  MoveL speed 30 mm/s, acceleration 50 mm/s^2 (useActiveTCP=true optimoveEnabled=false optiMoveSpeed=0.3 optiMoveAcceleration=0.09) feature=Base
    SuppressedNode
      Waypoint r1_ek_front: TCP in base x=439.065 y=405.452 z=65.996 mm, rx=2.3168 ry=2.0514 rz=0.0766 rad; joints [-187.962, -93.321, 143.386, -27.168, -1.131, -26.752] deg
    SuppressedNode
      Waypoint r1_ek_middle: TCP in base x=419.01 y=404.851 z=65.995 mm, rx=2.3096 ry=2.0447 rz=0.0891 rad; joints [-188.553, -97.485, 146.002, -33.769, -1.69, -19.324] deg
    SuppressedNode
      Waypoint r1_ek_middle2: TCP in base x=417.012 y=405.435 z=65.003 mm, rx=2.3169 ry=2.0513 rz=0.0766 rad; joints [-188.493, -97.025, 145.794, -33.21, -1.638, -19.415] deg
    SuppressedNode
      Waypoint r1_ek_bottom: TCP in base x=413.072 y=405.431 z=68 mm, rx=2.3168 ry=2.0513 rz=0.0767 rad; joints [-188.596, -97.887, 146.02, -33.517, -1.738, -18.475] deg
    SuppressedNode
      Waypoint r1_ek_end: TCP in base x=389.999 y=405.444 z=68.005 mm, rx=2.3169 ry=2.0514 rz=0.0766 rad; joints [-189.248, -101.07, 148.002, -36.337, -2.38, -14.447] deg
    Waypoint Variable (Variable): variable=ek_front
    Waypoint Variable (Variable): variable=ek_middle
    Waypoint Variable (Variable): variable=ek_middle2
    Waypoint Variable (Variable): variable=ek_bottom
    Waypoint Variable (Variable): variable=ek_end
  MoveJ speed 60 deg/s, acceleration 80 deg/s^2 (useActiveTCP=true optimoveEnabled=false optiMoveSpeed=0.3 optiMoveAcceleration=0.09) feature=Base
    SuppressedNode
      Waypoint r1_ek_oldhome: TCP in base x=397.38 y=356.254 z=319.821 mm, rx=2.3163 ry=2.0576 rz=0.0741 rad; joints [-198.126, -117.851, 133.303, -13.009, -11.422, -6.035] deg
    Waypoint Variable (Variable): variable=ek_oldhome
    'above waypoint is home'
  SuppressedNode
    SafeHome (positionOptionType=SPEED_AND_ACCELERATION speed=1.047198 acceleration=1.396263 nextMotionTime=2)
SubProgram Straight_Homing_Floor_2 (keepSynchronizedWithDisk=false) programFile=/programs/Straight Homing Floor 2.urp
  Set NoAction tcp=pretend_w_top
  'dummy move below for debug'
  SuppressedNode
    Folder dummy points
      MoveL speed 100 mm/s, acceleration 1200 mm/s^2 (useActiveTCP=true optimoveEnabled=false optiMoveSpeed=0.3 optiMoveAcceleration=0.09) feature=Base
        Waypoint tcp_l: TCP in base x=-1157.117 y=-14.284 z=-81.871 mm, rx=1.2641 ry=-1.1744 rz=-0.9868 rad; joints [-20.789, -44.61, 126.749, -78.291, 59.56, 3.601] deg; TCP offset x=0.14 y=-17.51 z=284 mm, rx=0 ry=0 rz=0 rad
        Waypoint tcp_r: TCP in base x=-1091.012 y=400.793 z=-81.871 mm, rx=1.2641 ry=-1.1744 rz=-0.9868 rad; joints [-50.03, -43.105, 118.828, -69.165, 30.433, -0.106] deg
      tcp_pose_left := tcp_l
      tcp_pose_right := tcp_r
  SuppressedNode
    SafeHome (positionOptionType=SPEED_AND_ACCELERATION speed=1.047198 acceleration=1.396263 nextMotionTime=2)
  SuppressedNode
    MoveJ speed 60 deg/s, acceleration 80 deg/s^2 (useActiveTCP=true optimoveEnabled=false optiMoveSpeed=0.3 optiMoveAcceleration=0.09) feature=Base
      Waypoint demo_point0: TCP in base x=-1268.829 y=243.799 z=397.866 mm, rx=1.3918 ry=-0.5735 rz=-1.0174 rad; joints [-39.169, -62.377, 106.188, -68.476, 20.677, 9.969] deg; TCP offset x=-1.032 y=-18.062 z=285.234 mm, rx=0 ry=0 rz=0 rad
  SuppressedNode
    MoveJ speed 60 deg/s, acceleration 80 deg/s^2 (useActiveTCP=true optimoveEnabled=false optiMoveSpeed=0.3 optiMoveAcceleration=0.09) feature=Base
      Waypoint Waypoint_1: TCP in base x=-589.354 y=-224.033 z=519.728 mm, rx=1.0077 ry=-1.3585 rz=-1.2216 rad; joints [24.032, -118.039, 143.045, -26.295, 122.645, 7.654] deg
      Waypoint Waypoint_2: TCP in base x=-1013.668 y=283.774 z=13.404 mm, rx=-0.1302 ry=-1.6605 rz=-0.1403 rad; joints [-36.803, -53.188, 133.142, -74.065, 63.057, 86.565] deg; TCP offset x=0 y=0 z=246 mm, rx=0 ry=0 rz=0 rad
  Wait Sleep waitTime=1
  SuppressedNode
    tp := get_actual_tcp_pose()
  Script file /programs/analyze_touchpoints.script
    | (same text as the earlier copy of this file)
  path_pre := get_straight_homing_pathpoints_floor(tcp_pose_left,tcp_pose_right)
  ph1 := path_pre[0]
  ph2 := path_pre[1]
  ph3 := path_pre[2]
  ph4 := path_pre[3]
  ph4a := p[ph4[0]+0.1,ph4[1],ph4[2],ph4[3],ph4[4],ph4[5]]
  MoveL speed 250 mm/s, acceleration 1200 mm/s^2 (useActiveTCP=true optimoveEnabled=false optiMoveSpeed=0.3 optiMoveAcceleration=0.09) feature=Base
    MoveDirectionNode (selectedDirection=XPlus)
      Until DISTANCE (allowActions=false deceleration=3 distanceNodeType=STOP) Distance=0.1; motionParameters(blendRadius=0)
  SuppressedNode
    MoveJ speed 60 deg/s, acceleration 80 deg/s^2 (useActiveTCP=true optimoveEnabled=false optiMoveSpeed=0.3 optiMoveAcceleration=0.09) feature=Base
      SuppressedNode
        Waypoint Waypoint_11: TCP in base x=-589.354 y=-454.462 z=658.693 mm, rx=1.8664 ry=-1.8664 rz=-0.5984 rad; joints [32.16, -93.601, 92.579, 59.83, 108.044, 27.179] deg; TCP offset x=-1.032 y=-18.062 z=285.234 mm, rx=0 ry=0 rz=0 rad
      Waypoint Waypoint_1: TCP in base x=-589.354 y=-224.033 z=519.728 mm, rx=1.0077 ry=-1.3585 rz=-1.2216 rad; joints [24.032, -118.039, 143.045, -26.295, 122.645, 7.654] deg
  MoveL speed 250 mm/s, acceleration 200 mm/s^2 (useActiveTCP=true optimoveEnabled=false optiMoveSpeed=0.3 optiMoveAcceleration=0.09) feature=Base
    Waypoint Variable (Variable): variable=ph2
  MoveL speed 20 mm/s, acceleration 100 mm/s^2 (useActiveTCP=true optimoveEnabled=false optiMoveSpeed=0.3 optiMoveAcceleration=0.09) feature=Base
    MoveDirectionNode (selectedDirection=XMinus)
      Until TOOL_CONTACT_DETECTION (allowActions=false retraction=0 decelerationAcceleration=3 decelerationAngularAcceleration=34.906585)
  p12 := get_actual_tcp_pose()
  MoveL speed 250 mm/s, acceleration 1200 mm/s^2 (useActiveTCP=true optimoveEnabled=false optiMoveSpeed=0.3 optiMoveAcceleration=0.09) feature=Base
    Waypoint Variable (Variable): variable=ph2
    Waypoint Variable (Variable): variable=ph1
  MoveL speed 20 mm/s, acceleration 100 mm/s^2 (useActiveTCP=true optimoveEnabled=false optiMoveSpeed=0.3 optiMoveAcceleration=0.09) feature=Base
    MoveDirectionNode (selectedDirection=XMinus)
      Until TOOL_CONTACT_DETECTION (allowActions=false retraction=0 decelerationAcceleration=3 decelerationAngularAcceleration=34.906585)
  SuppressedNode
    p13 := get_actual_tcp_pose()
  SuppressedNode
    MoveJ speed 60 deg/s, acceleration 80 deg/s^2 (useActiveTCP=true optimoveEnabled=false optiMoveSpeed=0.3 optiMoveAcceleration=0.09) feature=Base
      Waypoint Variable (Variable): variable(name=ph2up)
      Waypoint Variable (Variable): variable=ph3
  SuppressedNode
    MoveL speed 20 mm/s, acceleration 100 mm/s^2 (useActiveTCP=true optimoveEnabled=false optiMoveSpeed=0.3 optiMoveAcceleration=0.09) feature=Base
      MoveDirectionNode expression=[-1,-1.0,0.0]
        Until TOOL_CONTACT_DETECTION (allowActions=false retraction=0 decelerationAcceleration=3 decelerationAngularAcceleration=34.906585)
  p11 := get_actual_tcp_pose()
  MoveJ speed 60 deg/s, acceleration 80 deg/s^2 (useActiveTCP=true optimoveEnabled=false optiMoveSpeed=0.3 optiMoveAcceleration=0.09) feature=Base
    Waypoint Variable (Variable): variable=ph1
  SuppressedNode
    MoveJ speed 60 deg/s, acceleration 80 deg/s^2 (useActiveTCP=true optimoveEnabled=false optiMoveSpeed=0.3 optiMoveAcceleration=0.09) feature=Base
      Waypoint Variable (Variable): variable=ph1
  'start of new section'
  ph_back := p[-0.85,ph1[1],ph1[2],ph1[3],ph1[4],ph1[5]]
  'start spin'
  MoveL speed 250 mm/s, acceleration 1200 mm/s^2 (useActiveTCP=true optimoveEnabled=false optiMoveSpeed=0.3 optiMoveAcceleration=0.09) feature=Base
    Waypoint Variable (Variable): variable=ph_back
  MoveJ speed 60 deg/s, acceleration 80 deg/s^2 (useActiveTCP=true optimoveEnabled=false optiMoveSpeed=0.3 optiMoveAcceleration=0.09) feature=Base
    Waypoint Waypoint_1: TCP in base x=-859.669 y=-373.309 z=-21.871 mm, rx=1.209 ry=-1.209 rz=-1.209 rad; joints [20.633, -48.497, 142.021, -93.588, 110.677, -0.019] deg; TCP offset x=0.14 y=-17.51 z=284 mm, rx=0 ry=0 rz=0 rad
    SuppressedNode
      Waypoint Waypoint_3: TCP in base x=-859.669 y=-373.309 z=-21.871 mm, rx=0.2086 ry=-0.2089 rz=-1.5605 rad; joints [12.923, -3.882, 111.524, -182.82, 93.304, -12.474] deg
    Waypoint Waypoint_6: TCP in base x=-826.115 y=-379.848 z=-18.79 mm, rx=-0.0538 ry=-0.0807 rz=1.1703 rad; joints [11.816, -2.134, 104.65, -187.43, 91.002, 145.344] deg
  ph3a := p[ph3[0]+0.1,ph3[1],ph3[2],ph3[3],ph3[4],ph3[5]]
  MoveL speed 100 mm/s, acceleration 1200 mm/s^2 (useActiveTCP=true optimoveEnabled=false optiMoveSpeed=0.3 optiMoveAcceleration=0.09) feature=Base
    Waypoint Variable (Variable): variable=ph3a
    Waypoint Variable (Variable): variable=ph3
  Wait Sleep waitTime=0.5
  MoveL speed 20 mm/s, acceleration 100 mm/s^2 (useActiveTCP=true optimoveEnabled=false optiMoveSpeed=0.3 optiMoveAcceleration=0.09) feature=Base
    MoveDirectionNode (selectedDirection=ZPlus)
      Until TOOL_CONTACT_DETECTION (allowActions=false retraction=0 decelerationAcceleration=3 decelerationAngularAcceleration=34.906585)
  p21 := get_actual_tcp_pose()
  MoveL speed 100 mm/s, acceleration 1200 mm/s^2 (useActiveTCP=true optimoveEnabled=false optiMoveSpeed=0.3 optiMoveAcceleration=0.09) feature=Base
    Waypoint Variable (Variable): variable=ph3
    Waypoint Variable (Variable): variable=ph3a
    Waypoint Variable (Variable): variable=ph4a
    Waypoint Variable (Variable): variable=ph4
  Wait Sleep waitTime=0.5
  MoveL speed 20 mm/s, acceleration 100 mm/s^2 (useActiveTCP=true optimoveEnabled=false optiMoveSpeed=0.3 optiMoveAcceleration=0.09) feature=Base
    MoveDirectionNode (selectedDirection=ZPlus)
      Until TOOL_CONTACT_DETECTION (allowActions=false retraction=0 decelerationAcceleration=3 decelerationAngularAcceleration=34.906585)
  p22 := get_actual_tcp_pose()
  MoveL speed 100 mm/s, acceleration 1200 mm/s^2 (useActiveTCP=true optimoveEnabled=false optiMoveSpeed=0.3 optiMoveAcceleration=0.09) feature=Base
    Waypoint Variable (Variable): variable=ph4
    Waypoint Variable (Variable): variable=ph4a
  'retreat'
  MoveJ speed 60 deg/s, acceleration 80 deg/s^2 (useActiveTCP=true optimoveEnabled=false optiMoveSpeed=0.3 optiMoveAcceleration=0.09) feature=Base
    Waypoint Waypoint_8: TCP in base x=-528.587 y=855.731 z=-241.099 mm, rx=-0.0343 ry=-0.0418 rz=-1.096 rad; joints [-70.846, 12.059, 81.059, -180.218, 89.919, 98.05] deg
  MoveL speed 400 mm/s, acceleration 500 mm/s^2 (useActiveTCP=true optimoveEnabled=false optiMoveSpeed=0.3 optiMoveAcceleration=0.09) feature=Base
    SuppressedNode
      Waypoint Waypoint_20: TCP in base x=-528.587 y=855.731 z=735.19 mm, rx=-0.0343 ry=-0.0418 rz=-1.096 rad; joints [-70.811, -56.591, 119.754, -150.264, 89.964, 97.984] deg
    Waypoint Waypoint_24: TCP in base x=-131.14 y=855.731 z=156.011 mm, rx=-0.0343 ry=-0.0418 rz=-1.096 rad; joints [-96.36, -13.202, 116.888, -191.074, 88.653, 123.526] deg
    Waypoint Waypoint_23: TCP in base x=-59.798 y=855.731 z=735.19 mm, rx=-0.0343 ry=-0.0418 rz=-1.096 rad; joints [-101.249, -61.114, 131.529, -157.92, 88.47, 128.392] deg
  MoveJ speed 60 deg/s, acceleration 80 deg/s^2 (useActiveTCP=true optimoveEnabled=false optiMoveSpeed=0.3 optiMoveAcceleration=0.09) feature=Base
    Waypoint Waypoint_22: TCP in base x=624.813 y=687.862 z=772.423 mm, rx=0.1261 ry=2.3257 rz=2.0415 rad; joints [-174.51, -91.126, 100.648, 25.662, 12.935, -33.314] deg
  SafeHome (positionOptionType=SPEED_AND_ACCELERATION speed=1.047198 acceleration=1.396263 nextMotionTime=2)
  'end of new section'
  SuppressedNode
    MoveJ speed 60 deg/s, acceleration 80 deg/s^2 (useActiveTCP=true optimoveEnabled=false optiMoveSpeed=0.3 optiMoveAcceleration=0.09) feature=Base
      SuppressedNode
        Waypoint Waypoint_11: TCP in base x=-589.354 y=-454.462 z=658.693 mm, rx=1.8664 ry=-1.8664 rz=-0.5984 rad; joints [32.16, -93.601, 92.579, 59.83, 108.044, 27.179] deg; TCP offset x=-1.032 y=-18.062 z=285.234 mm, rx=0 ry=0 rz=0 rad
      Waypoint Waypoint_3: TCP in base x=-589.354 y=-224.033 z=519.728 mm, rx=1.0077 ry=-1.3585 rz=-1.2216 rad; joints [24.032, -118.039, 143.045, -26.295, 122.645, 7.654] deg
      SuppressedNode
        Waypoint Waypoint_3: TCP in base x=-1381.315 y=-113.246 z=483.261 mm, rx=0.347 ry=3.1015 rz=-0.0385 rad; joints [-4.848, -55.573, 57.279, 269.477, -88.568, -82.096] deg
      SuppressedNode
        Waypoint Waypoint_9: TCP in base x=-594.234 y=-418.092 z=645.151 mm, rx=0.1258 ry=-0.6986 rz=-0.4993 rad; joints [32.009, -82.779, 153.256, -126.399, 112.73, 35.158] deg
      SuppressedNode
        Waypoint Waypoint_6: TCP in base x=-563.856 y=-113.246 z=483.261 mm, rx=0.347 ry=3.1015 rz=-0.0385 rad; joints [-12.028, -113.359, 121.362, 263.351, -88.693, -89.284] deg
      SuppressedNode
        Waypoint Waypoint_15: TCP in base x=-841.932 y=-252.174 z=466.323 mm, rx=-0.1894 ry=-0.3294 rz=0.1013 rad; joints [8.59, -43.671, 136.758, -165.147, 102.406, 89.233] deg
      SuppressedNode
        Waypoint Waypoint_8: TCP in base x=-869.439 y=-409.581 z=418.615 mm, rx=0 ry=-0.0001 rz=0 rad; joints [12.101, -33.012, 119.104, -176.134, 89.938, 77.897] deg
      SuppressedNode
        Waypoint Waypoint_12: TCP in base x=-1028.087 y=-409.581 z=-52.555 mm, rx=0 ry=-0.0001 rz=0.7467 rad; joints [10.416, 0.258, 83.964, -174.263, 89.923, 122.381] deg
      SuppressedNode
        Waypoint Waypoint_13: TCP in base x=-867.034 y=98.846 z=-52.555 mm, rx=0 ry=-0.0001 rz=0.7467 rad; joints [-20.439, 1.166, 101.357, -192.565, 89.913, 153.243] deg
      Waypoint Waypoint_17: TCP in base x=-574.647 y=213.551 z=642.998 mm, rx=-0.2366 ry=-0.9664 rz=-0.9158 rad; joints [-39.25, -121.471, 159.271, -73.052, 92.515, 73.526] deg
      Waypoint Waypoint_16: TCP in base x=-343.952 y=632.142 z=615.175 mm, rx=-0.0259 ry=-0.0088 rz=-0.5675 rad; joints [-78.579, -51.22, 142.034, -179.331, 90.185, 136.06] deg
  SuppressedNode
    MoveJ speed 60 deg/s, acceleration 80 deg/s^2 (useActiveTCP=true optimoveEnabled=false optiMoveSpeed=0.3 optiMoveAcceleration=0.09) feature=Base
      Waypoint Waypoint_4: TCP in base x=-658.265 y=299.53 z=30.91 mm, rx=0.4268 ry=-1.6215 rz=0.4371 rad; joints [-77.363, -55.591, 142.792, -102.186, -19.322, 105.94] deg; TCP offset x=0 y=0 z=246 mm, rx=0 ry=0 rz=0 rad
      Waypoint Waypoint_5: TCP in base x=-448.863 y=524.6 z=-175.967 mm, rx=2.4733 ry=-1.8744 rz=0.2053 rad; joints [-65.056, -57.525, 139.86, -164.756, -91.924, 99.291] deg
      SuppressedNode
        Waypoint Waypoint_5: TCP in base x=-542.919 y=212.782 z=86.75 mm, rx=-0.746 ry=-1.5701 rz=-0.8083 rad; joints [-15.32, -63.738, 160.053, -88.648, -229.235, 89.501] deg
      Waypoint Waypoint_10: TCP in base x=-559.13 y=259.234 z=102.446 mm, rx=-0.8226 ry=-1.4861 rz=-0.8815 rad; joints [-31.871, -61.56, 166.811, -101.777, -239.831, 87.599] deg; TCP offset x=-1.157 y=-95.604 z=257.595 mm, rx=0 ry=0 rz=0 rad
  SuppressedNode
    Folder old
      MoveL speed 250 mm/s, acceleration 1200 mm/s^2 (useActiveTCP=true optimoveEnabled=false optiMoveSpeed=0.3 optiMoveAcceleration=0.09) feature=Base
        Waypoint Variable (Variable): variable=ph4a
        Waypoint Variable (Variable): variable=ph3
      MoveL speed 20 mm/s, acceleration 100 mm/s^2 (useActiveTCP=true optimoveEnabled=false optiMoveSpeed=0.3 optiMoveAcceleration=0.09) feature=Base
        MoveDirectionNode (selectedDirection=ZPlus)
          Until TOOL_CONTACT_DETECTION (allowActions=false retraction=0 decelerationAcceleration=3 decelerationAngularAcceleration=34.906585)
      p21 := get_actual_tcp_pose()
      MoveL speed 250 mm/s, acceleration 1200 mm/s^2 (useActiveTCP=true optimoveEnabled=false optiMoveSpeed=0.3 optiMoveAcceleration=0.09) feature=Base
        Waypoint Variable (Variable): variable=ph3
      MoveJ speed 60 deg/s, acceleration 80 deg/s^2 (useActiveTCP=true optimoveEnabled=false optiMoveSpeed=0.3 optiMoveAcceleration=0.09) feature=Base
        Waypoint Variable (Variable): variable=ph4
      MoveL speed 20 mm/s, acceleration 100 mm/s^2 (useActiveTCP=true optimoveEnabled=false optiMoveSpeed=0.3 optiMoveAcceleration=0.09) feature=Base
        MoveDirectionNode (selectedDirection=ZPlus)
          Until TOOL_CONTACT_DETECTION (allowActions=false retraction=0 decelerationAcceleration=3 decelerationAngularAcceleration=34.906585)
      p22 := get_actual_tcp_pose()
      MoveL speed 250 mm/s, acceleration 1200 mm/s^2 (useActiveTCP=true optimoveEnabled=false optiMoveSpeed=0.3 optiMoveAcceleration=0.09) feature=Base
        Waypoint Variable (Variable): variable=ph4
        Waypoint Variable (Variable): variable=ph4a
      MoveJ speed 60 deg/s, acceleration 80 deg/s^2 (useActiveTCP=true optimoveEnabled=false optiMoveSpeed=0.3 optiMoveAcceleration=0.09) feature=Base
        Waypoint Waypoint_16: TCP in base x=-343.952 y=632.142 z=615.175 mm, rx=-0.0259 ry=-0.0088 rz=-0.5675 rad; joints [-78.579, -51.22, 142.034, -179.331, 90.185, 136.06] deg; TCP offset x=-1.032 y=-18.062 z=285.234 mm, rx=0 ry=0 rz=0 rad
      SafeHome (positionOptionType=SPEED_AND_ACCELERATION speed=1.047198 acceleration=1.396263 nextMotionTime=2)
Thread Thread_1 (runOnlyOnce=true)
  Loop While (checkContinuously=false) expression=True
    If freedrive_m_var≟ True
      Script: freedrive_mode()
      free_dr_already := True
    Else 
      If free_dr_already
        Script: end_freedrive_mode()
    Script: sync()
SuppressedNode
  Thread Thread_2 (runOnlyOnce=false)
    Loop While (checkContinuously=false) expression=True
      If thread2trigger≟ True
        'do the dot extrude'
        Wait Sleep waitTime=5
        URCap WireTank Serial (WireTank Serial, WireTank, LLC) dataModel(byte_array=true, NODE_TITLE=Serial Bridge uR1, Command=[252,82,49], QUERY=false, OUTPUT_ENTRY=Static, Variable(key=OUTPUT_VARIABLE, variable(name=HwResp)))
        Wait Sleep waitTime=2
        URCap WireTank Serial (WireTank Serial, WireTank, LLC) dataModel(QUERY=false, NODE_TITLE=Serial Bridge uR0, Command=[252,82,48], byte_array=true, OUTPUT_ENTRY=Static, Variable(key=OUTPUT_VARIABLE, variable(name=HwResp)))
        thread2trigger := False
      Script: sync()
